// 40 Visualizations/Dialog/DIA_MANAGERCONFIG
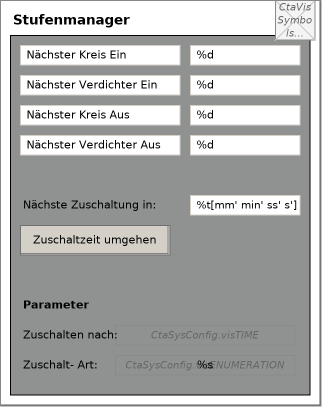
VISUALIZATION DIA_MANAGERCONFIG  // 322x407
VAR_IN_OUT
	{attribute 'VAR_IN_OUT_AS_POINTER'}
	MANAGER_DIA			:	MANAGER;
END_VAR
    RoundedRectangle (0,0 320x405)
    RoundedRectangle (10,35 300x360)
    Button (20,225 150x30), "Zuschaltzeit umgehen"
        toggle MANAGER_DIA.xResettReleaseLock_VIS
    Textfield (20,45 160x20), "Nächster Kreis Ein"
    Textfield (20,75 160x20), "Nächster Verdichter Ein"
    Textfield (20,135 160x20), "Nächster Verdichter Aus"
    Textfield (20,105 160x20), "Nächster Kreis Aus"
    Textfield (190,45 110x20), "%d", text variable: MANAGER_DIA.next_circuit_to_run_engine
    Textfield (190,75 110x20), "%d", text variable: MANAGER_DIA.next_engine_to_run
    Textfield (190,105 110x20), "%d", text variable: MANAGER_DIA.next_circuit_to_stopp_engine
    Textfield (190,135 110x20), "%d", text variable: MANAGER_DIA.next_engine_to_stopp
    Frame (115,325 180x20)
        shows CtaSysConfig.visTIME(visfbTIMEIn := MANAGER_DIA.scParameter.fbtZuschaltSperrzeit)
    Frame (115,355 180x20)
        shows CtaSysConfig.visENUMERATION(visfbENUIn := MANAGER_DIA.scParameter.fbiTypeOfEngineManagement)
    Label (20,325 150x20), "Zuschalten nach:"
    Label (20,355 150x20), "Zuschalt- Art:"
    Textfield (190,195 110x20), "%t[mm' min' ss' s']", text variable: (MANAGER_DIA.scParameter.fbtZuschaltSperrzeit.proValue - MANAGER_DIA.TP_ReleaseLock.ET)
    Textfield (20,195 160x20), "Nächste Zuschaltung in:"
    Textfield (20,295 160x20), "Parameter"
    Image (275,0 40x40), image: CtaVisSymbols.ImagePool.close_solo_black
        OnMouseClick:  Dialog=Current Dialog, Result=OK, NumpadKeypadSet=True
    Label (10,0 150x40), "Stufenmanager"
    Textfield (135,355 140x20), "%s", text list: 'TypeOfEngineManagement', text index: CtaSysConfig.fcGetEnumerationId(MANAGER_DIA.scParameter.fbiTypeOfEngineManagement)
END_VISUALIZATION

// 40 Visualizations/VIS_Manager_rEck
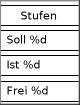
VISUALIZATION VIS_Manager_rEck  // 80x105
VAR_IN_OUT
	MANAGER_IN		:	MANAGER;
END_VAR
    Textfield (0,1 80x105)
    Textfield (0,6 78x20), "Stufen"
    Textfield (0,30 78x20), "Soll %d", text variable: MANAGER_IN.iRelease
    Textfield (0,55 78x20), "Ist %d", text variable: MANAGER_IN.iAcknowledged
    Textfield (0,81 78x20), "Frei %d", text variable: MANAGER_IN.iAvailableTemp
    Line (0,30) (79,30)
    Line (0,50) (79,50)
    Line (0,55) (79,55)
    Line (0,75) (79,75)
    Line (0,81) (79,81)
    Line (0,101) (79,101)
    Line (0,5) (79,5)
    Line (0,25) (79,25)
    Rectangle (0,0 80x105)
        OnMouseClick:  Dialog=DIA_MANAGERCONFIG, Parameters={MANAGER_DIA: MANAGER_IN}, Selected={0: }, OpenCentered=True
END_VISUALIZATION

// 40 Visualizations/VIS_Manager
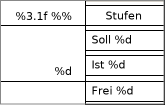
VISUALIZATION VIS_Manager  // 165x105
VAR_IN_OUT
	MANAGER_IN		:	MANAGER;
END_VAR
    Line (0,25) (157,25)
    Line (0,81) (158,81)
    Rectangle (15,65 60x13), "%d", text variable: MANAGER_IN.iRelease
    Rectangle (15,10 60x13), "%3.1f %%", text variable: MANAGER_IN.rRelease
    Frame (85,0 80x105)
        shows VIS_Manager_rEck(MANAGER_IN := MANAGER_IN)
END_VISUALIZATION

(* text list TypeOfEngineManagement (id | default | de | en | fr | it)
  0 | RUN 1BY1 |  |  |  | 
  1 | RUN EQUAL |  |  |  | 
   |  |  |  |  |  *)
